(* Logix 5000 project; controller cal1632 1756-L62 rev 16.20; software revision 16.05; part 16 of 61 *)
(* tags used below, declared in another part *)
   FAULT : BOOL;
   HMI : BOOL;
   p01r09_pb_global_reset : BOOL;
   p12_ai_exhaust_amps : REAL;
   p12_ai_exhaust_hz : REAL;
   p12_ai_exhaust_pct : REAL;
   p12_ai_exhaust_rpm : REAL;
   p12_ai_lfl : REAL;
   p12_ai_prs : REAL;
   p12_ai_recirc_amps : REAL;
   p12_ai_recirc_hz : REAL;
   p12_ai_recirc_pct : REAL;
   p12_ai_recirc_rpm : REAL;
   p12_ai_tc01 : REAL;
   p12_ai_tc02 : REAL;
   p12_ao_cv : REAL;
   p12_ao_exhaust_selected_speed : REAL;
   p12_ao_recirc_selected_speed : REAL;
   p12_di_burner_auto : BOOL;
   p12_di_burner_safeties_ok : BOOL;
   p12_di_door_open : BOOL;
   p12_di_exh : acs800_di_normal;
   p12_di_exh_fan_mtr_ts : BOOL;
   p12_di_exh_flow_ok : BOOL;
   p12_di_flame_failure : BOOL;
   p12_di_flame_on : BOOL;
   p12_di_fresh_air_clean : BOOL;
   p12_di_high_limit_temp_ok : BOOL;
   p12_di_recirc : acs800_di_normal;
   p12_di_recirc_fan_mtr_ts : BOOL;
   p12_di_recirc_flow_ok : BOOL;
   p12_di_sp00 : BOOL;
   p12_di_tc01_bo : BOOL;
   p12_di_tc02_bo : BOOL;
   p12_di_zone_air_clean : BOOL;
   p12_dint_to_hmi : DINT[16];
   p12_param_fast_to_soak : REAL;
   p12_param_lfl_hhl : REAL;
   p12_param_lfl_hl : REAL;
   p12_param_pid1_ff : REAL;
   p12_param_pid1_kd : REAL;
   p12_param_pid1_ki : REAL;
   p12_param_pid1_kp : REAL;
   p12_param_pid2_ff : REAL;
   p12_param_pid2_kd : REAL;
   p12_param_pid2_ki : REAL;
   p12_param_pid2_kp : REAL;
   p12_param_shutdown_temp : REAL;
   p12_param_soak_to_fast : REAL;
   p12_param_tc01_dev : REAL;
   p12_param_tc01_hl : REAL;
   p12_param_tc01z : REAL;
   p12_param_tc02z : REAL;
   p12_param_zone_pressure : REAL;
   p12_real_to_hmi : REAL[112];
   p12r05 : routine;
   p12r05_exh_status : DINT;
   p12r05_recirc_status : DINT;
   p12r05_Temp_ctl_status : DINT;
   p12r05_timer_fault : TIMER[4];
   p12r05_timer_warning : TIMER[4];
   p12r06 : routine;
   p12r06_timer_fault : TIMER[4];
   p12r06_timer_warning : TIMER[4];
   p12r07 : routine;
   p12r07_timer_fault : TIMER[4];
   p12r07_timer_warning : TIMER[4];
   p12r20 : routine;
   p12r20_state : DINT;
   p12r20_status : DINT;
   p12r30 : routine;
   p12r30_cv_man_sp : REAL;
   p12r30_permissive_run : BOOL;
   p12r30_pid_temp : PID;
   p12r30_pid_temp_pv : REAL;
   p12r30_pid_temp_sp : REAL;
   p12r30_request_heat : BOOL;
   p12r30_request_manual : BOOL;
   p12r30_vfds_ready : BOOL;
   p12r31 : routine;
   p12r31_request_auto_run : BOOL;
   p12r31_request_auto_stop : BOOL;
   p12r31_vfd_stopped : BOOL;
   p12r32 : routine;
   p12r32_request_auto_run : BOOL;
   p12r32_request_auto_stop : BOOL;
   p12r32_vfd_stopped : BOOL;
(* P12_Zone_2, continued *)

ROUTINE R05_Dint_to_HMI   (* ladder *)
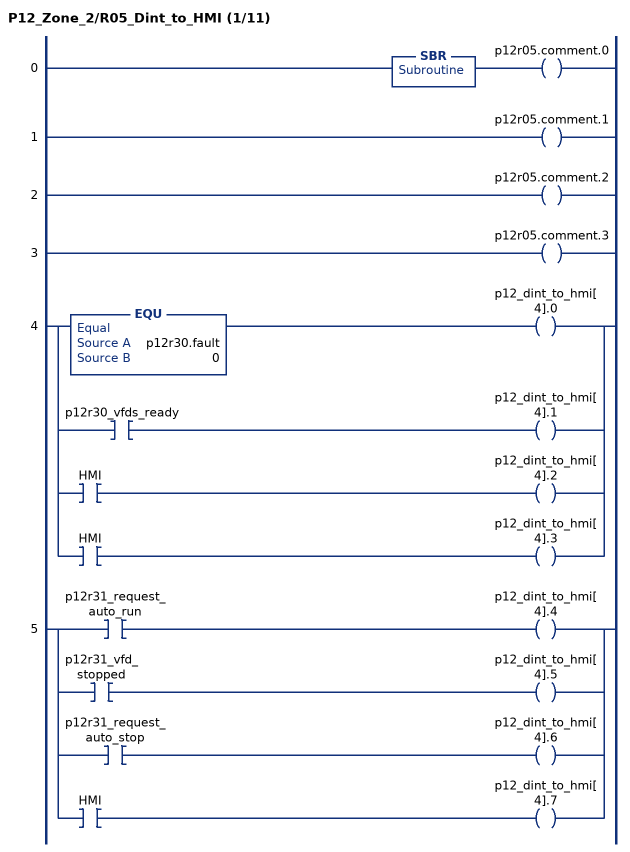
   0: SBR()OTE(p12r05.comment.0);
   1: OTE(p12r05.comment.1);
   2: OTE(p12r05.comment.2);
   3: OTE(p12r05.comment.3);
   4: [EQU(p12r30.fault,0) OTE(p12_dint_to_hmi[4].0) ,XIC(p12r30_vfds_ready) OTE(p12_dint_to_hmi[4].1) ,XIC(HMI) OTE(p12_dint_to_hmi[4].2) ,XIC(HMI) OTE(p12_dint_to_hmi[4].3) ];
   5: [XIC(p12r31_request_auto_run) OTE(p12_dint_to_hmi[4].4) ,XIC(p12r31_vfd_stopped) OTE(p12_dint_to_hmi[4].5) ,XIC(p12r31_request_auto_stop) OTE(p12_dint_to_hmi[4].6) ,XIC(HMI) OTE(p12_dint_to_hmi[4].7) ];
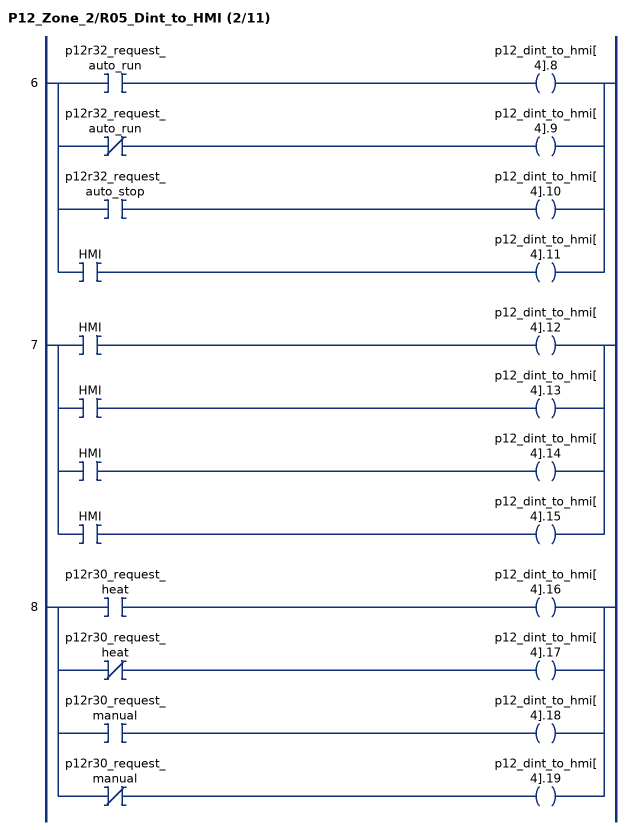
   6: [XIC(p12r32_request_auto_run) OTE(p12_dint_to_hmi[4].8) ,XIO(p12r32_request_auto_run) OTE(p12_dint_to_hmi[4].9) ,XIC(p12r32_request_auto_stop) OTE(p12_dint_to_hmi[4].10) ,XIC(HMI) OTE(p12_dint_to_hmi[4].11) ];
   7: [XIC(HMI) OTE(p12_dint_to_hmi[4].12) ,XIC(HMI) OTE(p12_dint_to_hmi[4].13) ,XIC(HMI) OTE(p12_dint_to_hmi[4].14) ,XIC(HMI) OTE(p12_dint_to_hmi[4].15) ];
   8: [XIC(p12r30_request_heat) OTE(p12_dint_to_hmi[4].16) ,XIO(p12r30_request_heat) OTE(p12_dint_to_hmi[4].17) ,XIC(p12r30_request_manual) OTE(p12_dint_to_hmi[4].18) ,XIO(p12r30_request_manual) OTE(p12_dint_to_hmi[4].19) ];
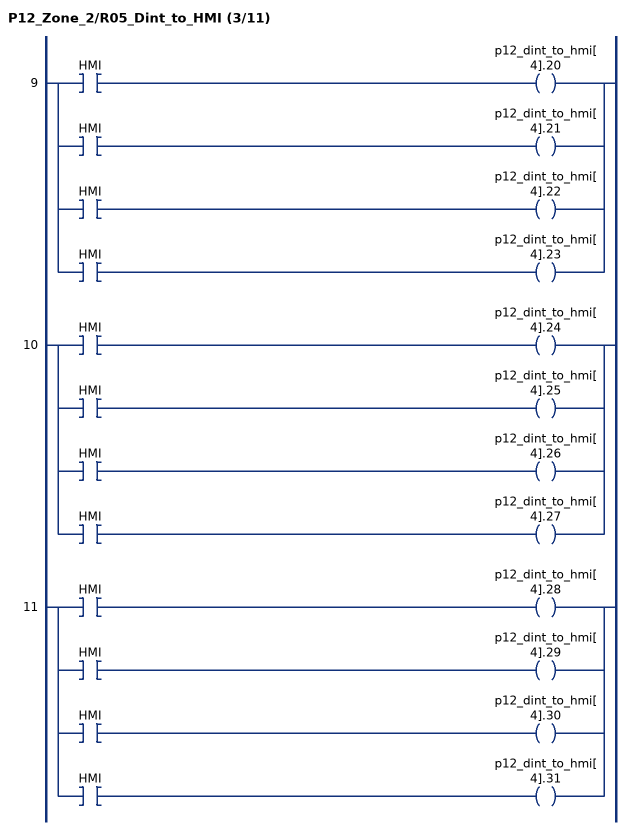
   9: [XIC(HMI) OTE(p12_dint_to_hmi[4].20) ,XIC(HMI) OTE(p12_dint_to_hmi[4].21) ,XIC(HMI) OTE(p12_dint_to_hmi[4].22) ,XIC(HMI) OTE(p12_dint_to_hmi[4].23) ];
   10: [XIC(HMI) OTE(p12_dint_to_hmi[4].24) ,XIC(HMI) OTE(p12_dint_to_hmi[4].25) ,XIC(HMI) OTE(p12_dint_to_hmi[4].26) ,XIC(HMI) OTE(p12_dint_to_hmi[4].27) ];
   11: [XIC(HMI) OTE(p12_dint_to_hmi[4].28) ,XIC(HMI) OTE(p12_dint_to_hmi[4].29) ,XIC(HMI) OTE(p12_dint_to_hmi[4].30) ,XIC(HMI) OTE(p12_dint_to_hmi[4].31) ];
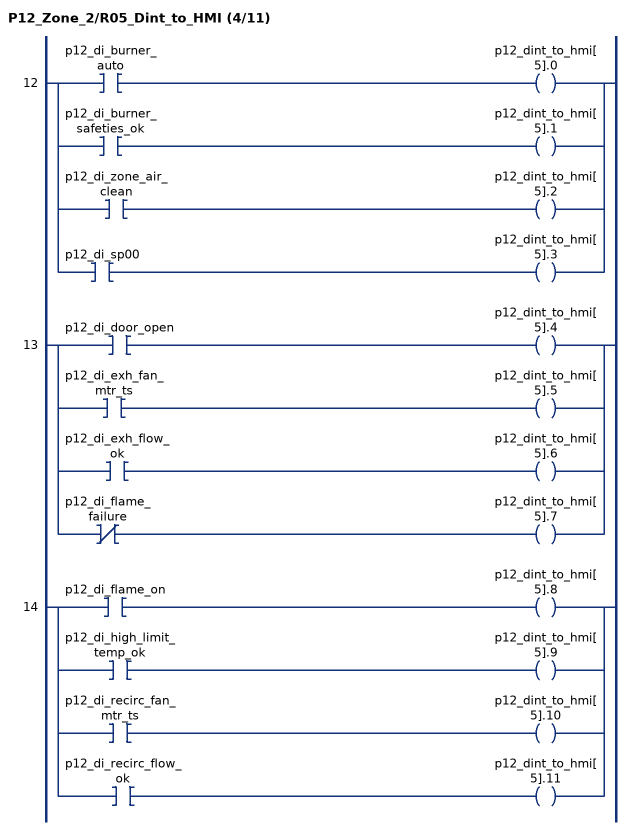
   12: [XIC(p12_di_burner_auto) OTE(p12_dint_to_hmi[5].0) ,XIC(p12_di_burner_safeties_ok) OTE(p12_dint_to_hmi[5].1) ,XIC(p12_di_zone_air_clean) OTE(p12_dint_to_hmi[5].2) ,XIC(p12_di_sp00) OTE(p12_dint_to_hmi[5].3) ];
   13: [XIC(p12_di_door_open) OTE(p12_dint_to_hmi[5].4) ,XIC(p12_di_exh_fan_mtr_ts) OTE(p12_dint_to_hmi[5].5) ,XIC(p12_di_exh_flow_ok) OTE(p12_dint_to_hmi[5].6) ,XIO(p12_di_flame_failure) OTE(p12_dint_to_hmi[5].7) ];
   14: [XIC(p12_di_flame_on) OTE(p12_dint_to_hmi[5].8) ,XIC(p12_di_high_limit_temp_ok) OTE(p12_dint_to_hmi[5].9) ,XIC(p12_di_recirc_fan_mtr_ts) OTE(p12_dint_to_hmi[5].10) ,XIC(p12_di_recirc_flow_ok) OTE(p12_dint_to_hmi[5].11) ];
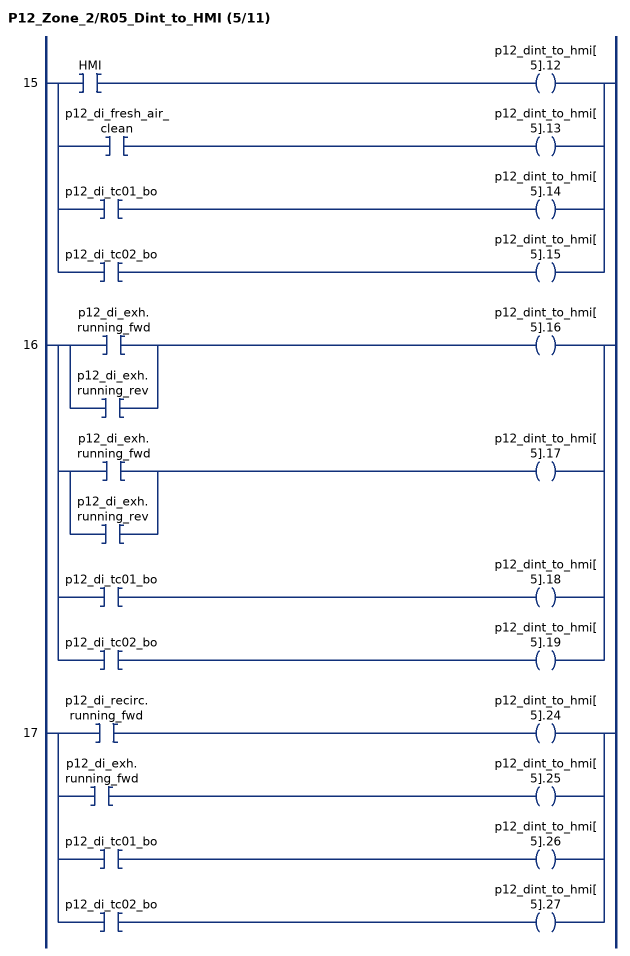
   15: [XIC(HMI) OTE(p12_dint_to_hmi[5].12) ,XIC(p12_di_fresh_air_clean) OTE(p12_dint_to_hmi[5].13) ,XIC(p12_di_tc01_bo) OTE(p12_dint_to_hmi[5].14) ,XIC(p12_di_tc02_bo) OTE(p12_dint_to_hmi[5].15) ];
   16: [[XIC(p12_di_exh.running_fwd) ,XIC(p12_di_exh.running_rev) ] OTE(p12_dint_to_hmi[5].16) ,[XIC(p12_di_exh.running_fwd) ,XIC(p12_di_exh.running_rev) ] OTE(p12_dint_to_hmi[5].17) ,XIC(p12_di_tc01_bo) OTE(p12_dint_to_hmi[5].18) ,XIC(p12_di_tc02_bo) OTE(p12_dint_to_hmi[5].19) ];
   17: [XIC(p12_di_recirc.running_fwd) OTE(p12_dint_to_hmi[5].24) ,XIC(p12_di_exh.running_fwd) OTE(p12_dint_to_hmi[5].25) ,XIC(p12_di_tc01_bo) OTE(p12_dint_to_hmi[5].26) ,XIC(p12_di_tc02_bo) OTE(p12_dint_to_hmi[5].27) ];
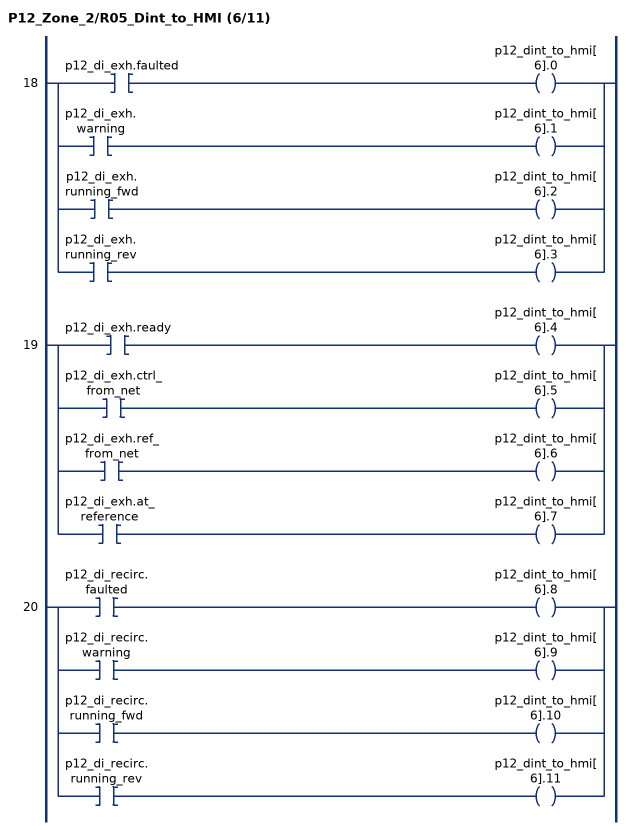
   18: [XIC(p12_di_exh.faulted) OTE(p12_dint_to_hmi[6].0) ,XIC(p12_di_exh.warning) OTE(p12_dint_to_hmi[6].1) ,XIC(p12_di_exh.running_fwd) OTE(p12_dint_to_hmi[6].2) ,XIC(p12_di_exh.running_rev) OTE(p12_dint_to_hmi[6].3) ];
   19: [XIC(p12_di_exh.ready) OTE(p12_dint_to_hmi[6].4) ,XIC(p12_di_exh.ctrl_from_net) OTE(p12_dint_to_hmi[6].5) ,XIC(p12_di_exh.ref_from_net) OTE(p12_dint_to_hmi[6].6) ,XIC(p12_di_exh.at_reference) OTE(p12_dint_to_hmi[6].7) ];
   20: [XIC(p12_di_recirc.faulted) OTE(p12_dint_to_hmi[6].8) ,XIC(p12_di_recirc.warning) OTE(p12_dint_to_hmi[6].9) ,XIC(p12_di_recirc.running_fwd) OTE(p12_dint_to_hmi[6].10) ,XIC(p12_di_recirc.running_rev) OTE(p12_dint_to_hmi[6].11) ];
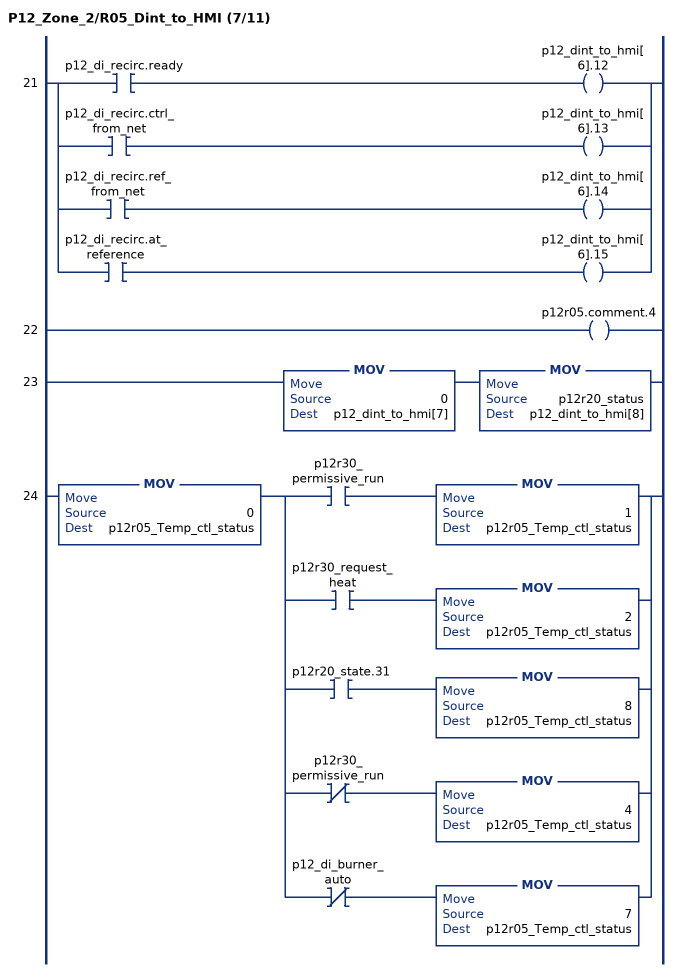
   21: [XIC(p12_di_recirc.ready) OTE(p12_dint_to_hmi[6].12) ,XIC(p12_di_recirc.ctrl_from_net) OTE(p12_dint_to_hmi[6].13) ,XIC(p12_di_recirc.ref_from_net) OTE(p12_dint_to_hmi[6].14) ,XIC(p12_di_recirc.at_reference) OTE(p12_dint_to_hmi[6].15) ];
   22: OTE(p12r05.comment.4);
   23: MOV(0,p12_dint_to_hmi[7])MOV(p12r20_status,p12_dint_to_hmi[8]);
   24: MOV(0,p12r05_Temp_ctl_status)[XIC(p12r30_permissive_run) MOV(1,p12r05_Temp_ctl_status) ,XIC(p12r30_request_heat) MOV(2,p12r05_Temp_ctl_status) ,XIC(p12r20_state.31) MOV(8,p12r05_Temp_ctl_status) ,XIO(p12r30_permissive_run) MOV(4,p12r05_Temp_ctl_status) ,XIO(p12_di_burner_auto) MOV(7,p12r05_Temp_ctl_status) ];
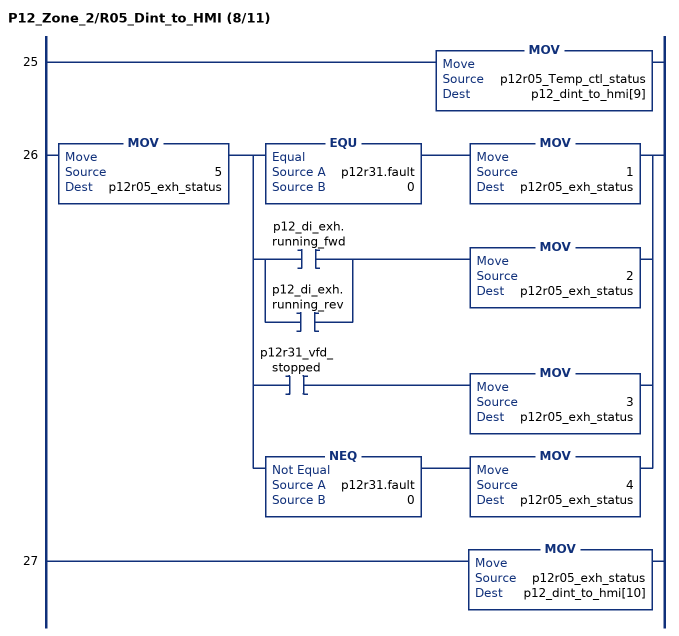
   25: MOV(p12r05_Temp_ctl_status,p12_dint_to_hmi[9]);
   26: MOV(5,p12r05_exh_status)[EQU(p12r31.fault,0) MOV(1,p12r05_exh_status) ,[XIC(p12_di_exh.running_fwd) ,XIC(p12_di_exh.running_rev) ] MOV(2,p12r05_exh_status) ,XIC(p12r31_vfd_stopped) MOV(3,p12r05_exh_status) ,NEQ(p12r31.fault,0) MOV(4,p12r05_exh_status) ];
   27: MOV(p12r05_exh_status,p12_dint_to_hmi[10]);
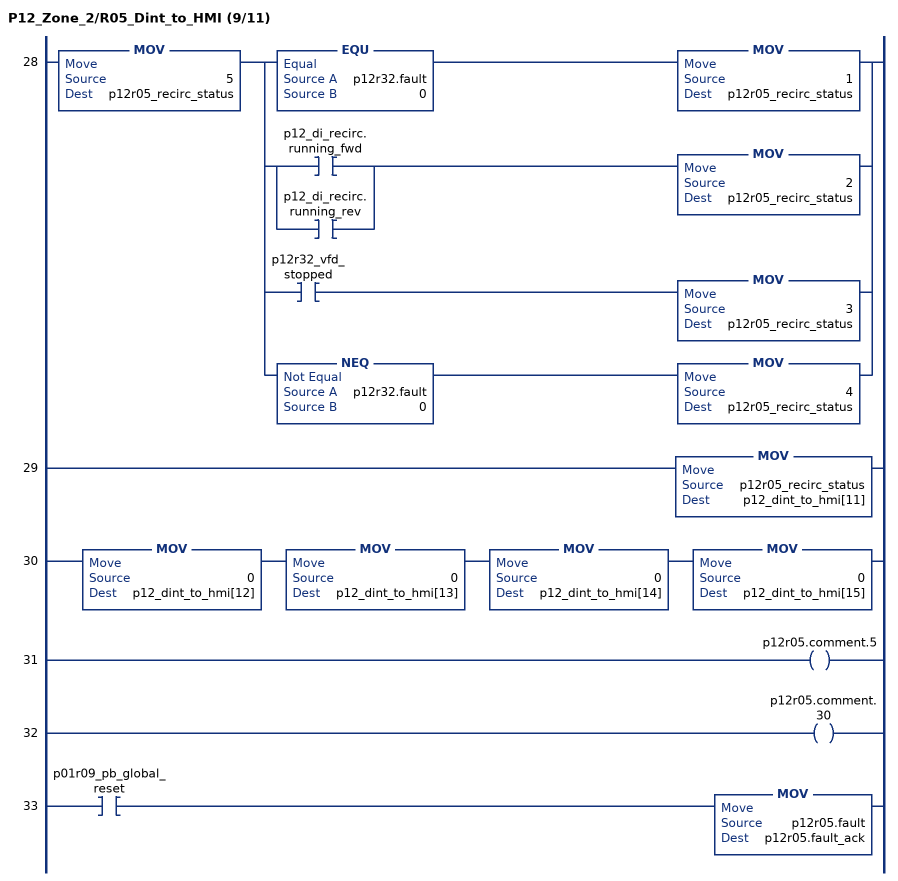
   28: MOV(5,p12r05_recirc_status)[EQU(p12r32.fault,0) MOV(1,p12r05_recirc_status) ,[XIC(p12_di_recirc.running_fwd) ,XIC(p12_di_recirc.running_rev) ] MOV(2,p12r05_recirc_status) ,XIC(p12r32_vfd_stopped) MOV(3,p12r05_recirc_status) ,NEQ(p12r32.fault,0) MOV(4,p12r05_recirc_status) ];
   29: MOV(p12r05_recirc_status,p12_dint_to_hmi[11]);
   30: MOV(0,p12_dint_to_hmi[12])MOV(0,p12_dint_to_hmi[13])MOV(0,p12_dint_to_hmi[14])MOV(0,p12_dint_to_hmi[15]);
   31: OTE(p12r05.comment.5);
   32: OTE(p12r05.comment.30);
   33: XIC(p01r09_pb_global_reset)MOV(p12r05.fault,p12r05.fault_ack);
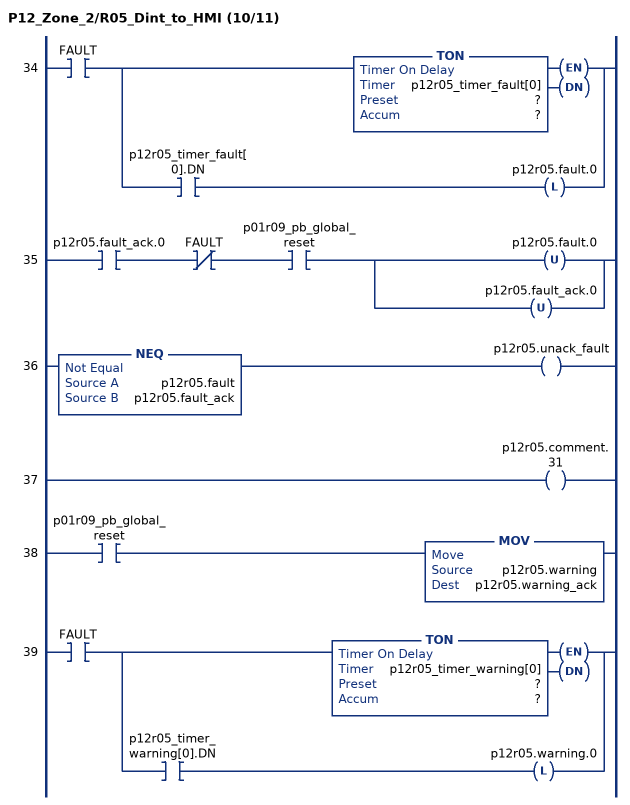
   34: XIC(FAULT)[TON(p12r05_timer_fault[0],?,?) ,XIC(p12r05_timer_fault[0].DN) OTL(p12r05.fault.0) ];
   35: XIC(p12r05.fault_ack.0)XIO(FAULT)XIC(p01r09_pb_global_reset)[OTU(p12r05.fault.0) ,OTU(p12r05.fault_ack.0) ];
   36: NEQ(p12r05.fault,p12r05.fault_ack)OTE(p12r05.unack_fault);
   37: OTE(p12r05.comment.31);
   38: XIC(p01r09_pb_global_reset)MOV(p12r05.warning,p12r05.warning_ack);
   39: XIC(FAULT)[TON(p12r05_timer_warning[0],?,?) ,XIC(p12r05_timer_warning[0].DN) OTL(p12r05.warning.0) ];
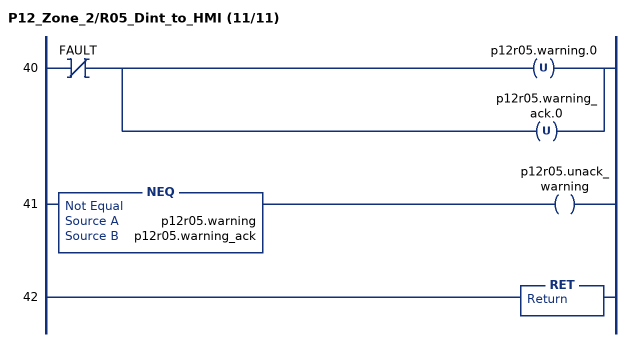
   40: XIO(FAULT)[OTU(p12r05.warning.0) ,OTU(p12r05.warning_ack.0) ];
   41: NEQ(p12r05.warning,p12r05.warning_ack)OTE(p12r05.unack_warning);
   42: RET();
END_ROUTINE

ROUTINE R06_Real_to_HMI   (* ladder *)
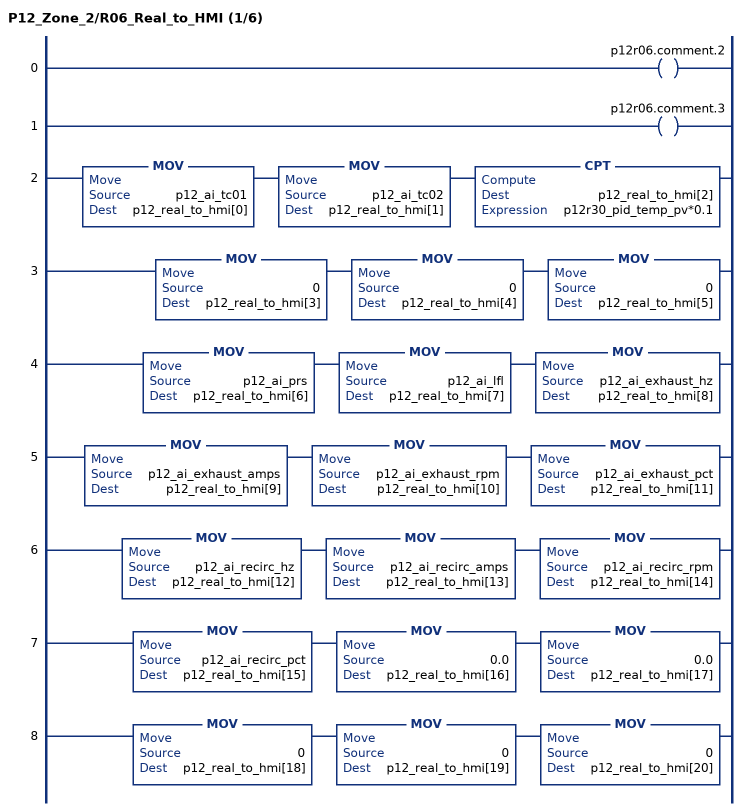
   0: OTE(p12r06.comment.2);
   1: OTE(p12r06.comment.3);
   2: MOV(p12_ai_tc01,p12_real_to_hmi[0])MOV(p12_ai_tc02,p12_real_to_hmi[1])CPT(p12_real_to_hmi[2],p12r30_pid_temp_pv*0.1);
   3: MOV(0,p12_real_to_hmi[3])MOV(0,p12_real_to_hmi[4])MOV(0,p12_real_to_hmi[5]);
   4: MOV(p12_ai_prs,p12_real_to_hmi[6])MOV(p12_ai_lfl,p12_real_to_hmi[7])MOV(p12_ai_exhaust_hz,p12_real_to_hmi[8]);
   5: MOV(p12_ai_exhaust_amps,p12_real_to_hmi[9])MOV(p12_ai_exhaust_rpm,p12_real_to_hmi[10])MOV(p12_ai_exhaust_pct,p12_real_to_hmi[11]);
   6: MOV(p12_ai_recirc_hz,p12_real_to_hmi[12])MOV(p12_ai_recirc_amps,p12_real_to_hmi[13])MOV(p12_ai_recirc_rpm,p12_real_to_hmi[14]);
   7: MOV(p12_ai_recirc_pct,p12_real_to_hmi[15])MOV(0.0,p12_real_to_hmi[16])MOV(0.0,p12_real_to_hmi[17]);
   8: MOV(0,p12_real_to_hmi[18])MOV(0,p12_real_to_hmi[19])MOV(0,p12_real_to_hmi[20]);
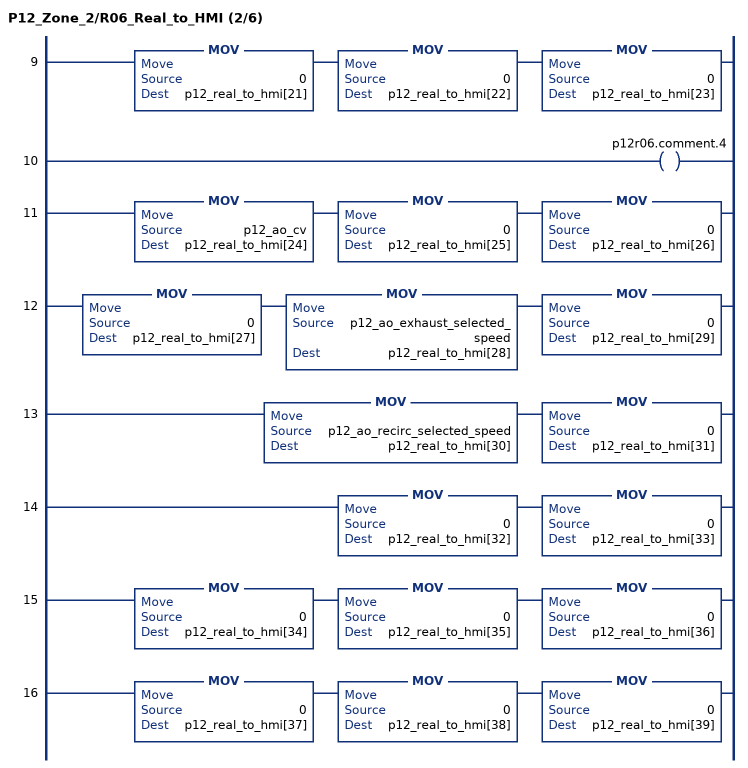
   9: MOV(0,p12_real_to_hmi[21])MOV(0,p12_real_to_hmi[22])MOV(0,p12_real_to_hmi[23]);
   10: OTE(p12r06.comment.4);
   11: MOV(p12_ao_cv,p12_real_to_hmi[24])MOV(0,p12_real_to_hmi[25])MOV(0,p12_real_to_hmi[26]);
   12: MOV(0,p12_real_to_hmi[27])MOV(p12_ao_exhaust_selected_speed,p12_real_to_hmi[28])MOV(0,p12_real_to_hmi[29]);
   13: MOV(p12_ao_recirc_selected_speed,p12_real_to_hmi[30])MOV(0,p12_real_to_hmi[31]);
   14: MOV(0,p12_real_to_hmi[32])MOV(0,p12_real_to_hmi[33]);
   15: MOV(0,p12_real_to_hmi[34])MOV(0,p12_real_to_hmi[35])MOV(0,p12_real_to_hmi[36]);
   16: MOV(0,p12_real_to_hmi[37])MOV(0,p12_real_to_hmi[38])MOV(0,p12_real_to_hmi[39]);
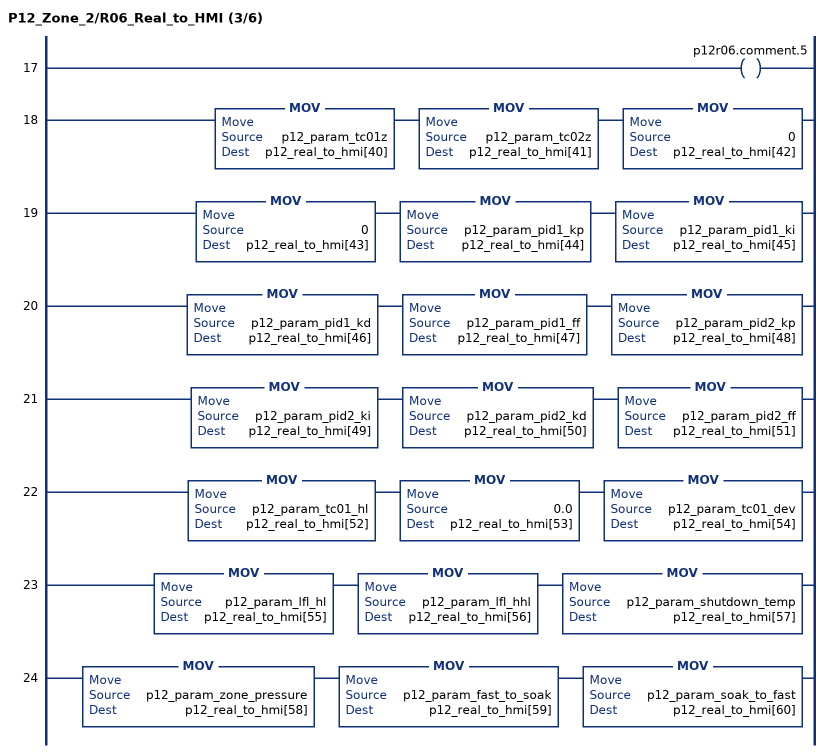
   17: OTE(p12r06.comment.5);
   18: MOV(p12_param_tc01z,p12_real_to_hmi[40])MOV(p12_param_tc02z,p12_real_to_hmi[41])MOV(0,p12_real_to_hmi[42]);
   19: MOV(0,p12_real_to_hmi[43])MOV(p12_param_pid1_kp,p12_real_to_hmi[44])MOV(p12_param_pid1_ki,p12_real_to_hmi[45]);
   20: MOV(p12_param_pid1_kd,p12_real_to_hmi[46])MOV(p12_param_pid1_ff,p12_real_to_hmi[47])MOV(p12_param_pid2_kp,p12_real_to_hmi[48]);
   21: MOV(p12_param_pid2_ki,p12_real_to_hmi[49])MOV(p12_param_pid2_kd,p12_real_to_hmi[50])MOV(p12_param_pid2_ff,p12_real_to_hmi[51]);
   22: MOV(p12_param_tc01_hl,p12_real_to_hmi[52])MOV(0.0,p12_real_to_hmi[53])MOV(p12_param_tc01_dev,p12_real_to_hmi[54]);
   23: MOV(p12_param_lfl_hl,p12_real_to_hmi[55])MOV(p12_param_lfl_hhl,p12_real_to_hmi[56])MOV(p12_param_shutdown_temp,p12_real_to_hmi[57]);
   24: MOV(p12_param_zone_pressure,p12_real_to_hmi[58])MOV(p12_param_fast_to_soak,p12_real_to_hmi[59])MOV(p12_param_soak_to_fast,p12_real_to_hmi[60]);
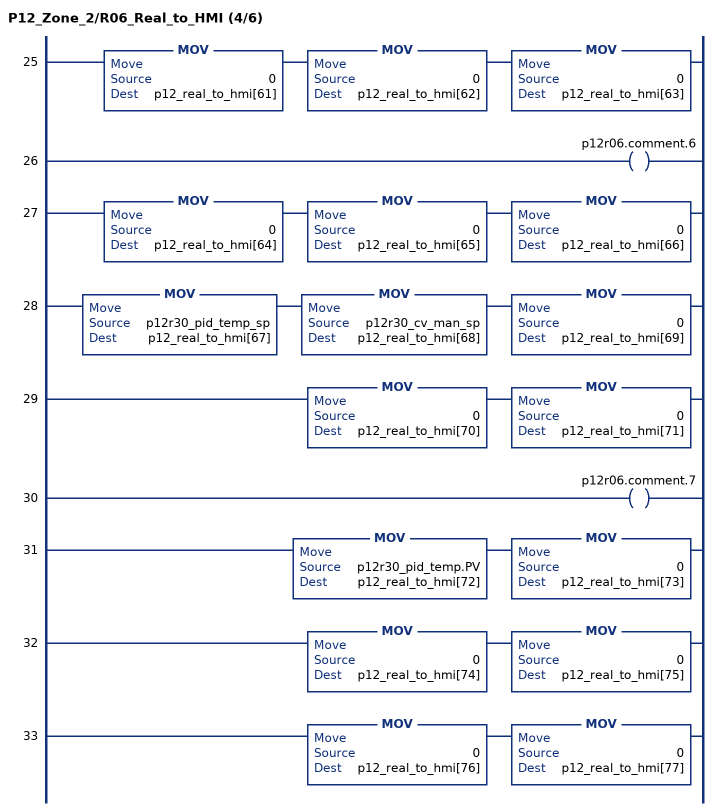
   25: MOV(0,p12_real_to_hmi[61])MOV(0,p12_real_to_hmi[62])MOV(0,p12_real_to_hmi[63]);
   26: OTE(p12r06.comment.6);
   27: MOV(0,p12_real_to_hmi[64])MOV(0,p12_real_to_hmi[65])MOV(0,p12_real_to_hmi[66]);
   28: MOV(p12r30_pid_temp_sp,p12_real_to_hmi[67])MOV(p12r30_cv_man_sp,p12_real_to_hmi[68])MOV(0,p12_real_to_hmi[69]);
   29: MOV(0,p12_real_to_hmi[70])MOV(0,p12_real_to_hmi[71]);
   30: OTE(p12r06.comment.7);
   31: MOV(p12r30_pid_temp.PV,p12_real_to_hmi[72])MOV(0,p12_real_to_hmi[73]);
   32: MOV(0,p12_real_to_hmi[74])MOV(0,p12_real_to_hmi[75]);
   33: MOV(0,p12_real_to_hmi[76])MOV(0,p12_real_to_hmi[77]);
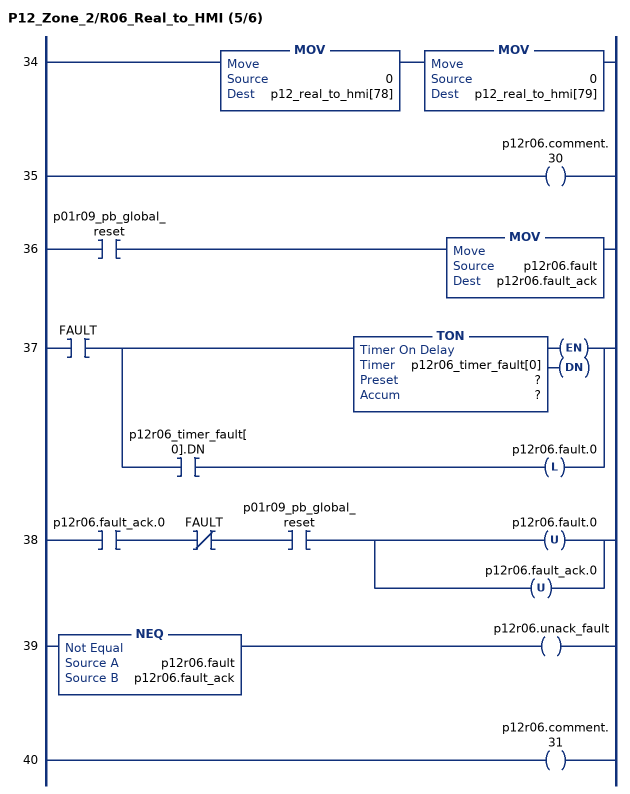
   34: MOV(0,p12_real_to_hmi[78])MOV(0,p12_real_to_hmi[79]);
   35: OTE(p12r06.comment.30);
   36: XIC(p01r09_pb_global_reset)MOV(p12r06.fault,p12r06.fault_ack);
   37: XIC(FAULT)[TON(p12r06_timer_fault[0],?,?) ,XIC(p12r06_timer_fault[0].DN) OTL(p12r06.fault.0) ];
   38: XIC(p12r06.fault_ack.0)XIO(FAULT)XIC(p01r09_pb_global_reset)[OTU(p12r06.fault.0) ,OTU(p12r06.fault_ack.0) ];
   39: NEQ(p12r06.fault,p12r06.fault_ack)OTE(p12r06.unack_fault);
   40: OTE(p12r06.comment.31);
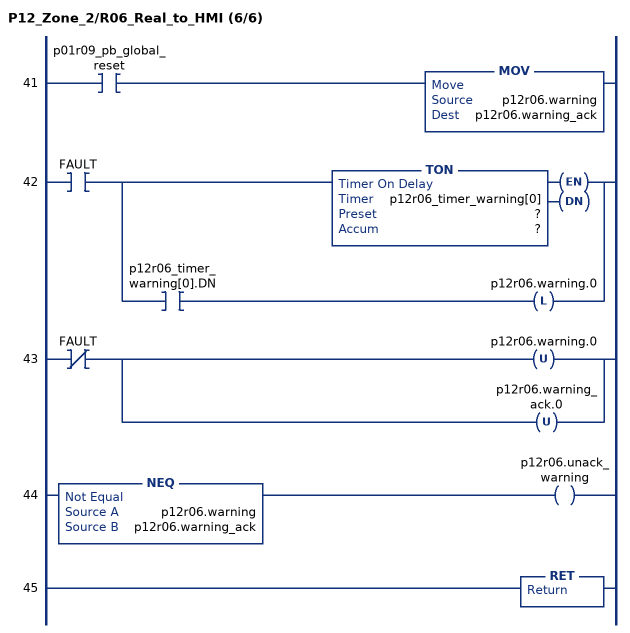
   41: XIC(p01r09_pb_global_reset)MOV(p12r06.warning,p12r06.warning_ack);
   42: XIC(FAULT)[TON(p12r06_timer_warning[0],?,?) ,XIC(p12r06_timer_warning[0].DN) OTL(p12r06.warning.0) ];
   43: XIO(FAULT)[OTU(p12r06.warning.0) ,OTU(p12r06.warning_ack.0) ];
   44: NEQ(p12r06.warning,p12r06.warning_ack)OTE(p12r06.unack_warning);
   45: RET();
END_ROUTINE

ROUTINE R07_Alarms   (* ladder *)
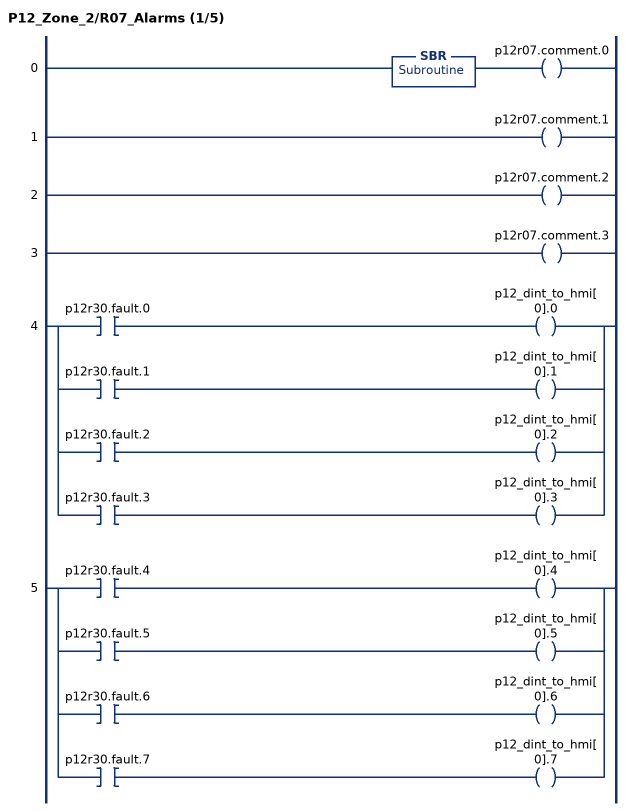
   0: SBR()OTE(p12r07.comment.0);
   1: OTE(p12r07.comment.1);
   2: OTE(p12r07.comment.2);
   3: OTE(p12r07.comment.3);
   4: [XIC(p12r30.fault.0) OTE(p12_dint_to_hmi[0].0) ,XIC(p12r30.fault.1) OTE(p12_dint_to_hmi[0].1) ,XIC(p12r30.fault.2) OTE(p12_dint_to_hmi[0].2) ,XIC(p12r30.fault.3) OTE(p12_dint_to_hmi[0].3) ];
   5: [XIC(p12r30.fault.4) OTE(p12_dint_to_hmi[0].4) ,XIC(p12r30.fault.5) OTE(p12_dint_to_hmi[0].5) ,XIC(p12r30.fault.6) OTE(p12_dint_to_hmi[0].6) ,XIC(p12r30.fault.7) OTE(p12_dint_to_hmi[0].7) ];
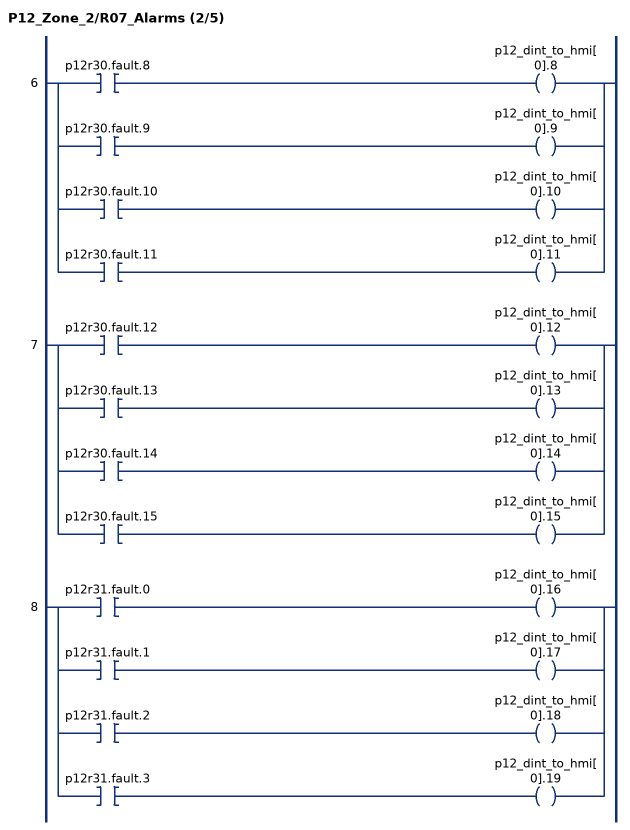
   6: [XIC(p12r30.fault.8) OTE(p12_dint_to_hmi[0].8) ,XIC(p12r30.fault.9) OTE(p12_dint_to_hmi[0].9) ,XIC(p12r30.fault.10) OTE(p12_dint_to_hmi[0].10) ,XIC(p12r30.fault.11) OTE(p12_dint_to_hmi[0].11) ];
   7: [XIC(p12r30.fault.12) OTE(p12_dint_to_hmi[0].12) ,XIC(p12r30.fault.13) OTE(p12_dint_to_hmi[0].13) ,XIC(p12r30.fault.14) OTE(p12_dint_to_hmi[0].14) ,XIC(p12r30.fault.15) OTE(p12_dint_to_hmi[0].15) ];
   8: [XIC(p12r31.fault.0) OTE(p12_dint_to_hmi[0].16) ,XIC(p12r31.fault.1) OTE(p12_dint_to_hmi[0].17) ,XIC(p12r31.fault.2) OTE(p12_dint_to_hmi[0].18) ,XIC(p12r31.fault.3) OTE(p12_dint_to_hmi[0].19) ];
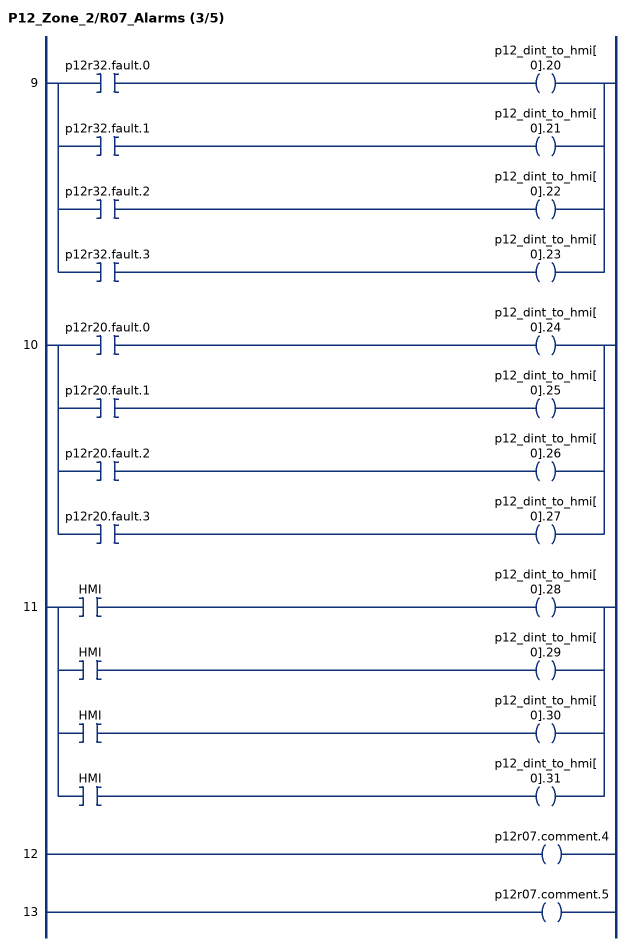
   9: [XIC(p12r32.fault.0) OTE(p12_dint_to_hmi[0].20) ,XIC(p12r32.fault.1) OTE(p12_dint_to_hmi[0].21) ,XIC(p12r32.fault.2) OTE(p12_dint_to_hmi[0].22) ,XIC(p12r32.fault.3) OTE(p12_dint_to_hmi[0].23) ];
   10: [XIC(p12r20.fault.0) OTE(p12_dint_to_hmi[0].24) ,XIC(p12r20.fault.1) OTE(p12_dint_to_hmi[0].25) ,XIC(p12r20.fault.2) OTE(p12_dint_to_hmi[0].26) ,XIC(p12r20.fault.3) OTE(p12_dint_to_hmi[0].27) ];
   11: [XIC(HMI) OTE(p12_dint_to_hmi[0].28) ,XIC(HMI) OTE(p12_dint_to_hmi[0].29) ,XIC(HMI) OTE(p12_dint_to_hmi[0].30) ,XIC(HMI) OTE(p12_dint_to_hmi[0].31) ];
   12: OTE(p12r07.comment.4);
   13: OTE(p12r07.comment.5);
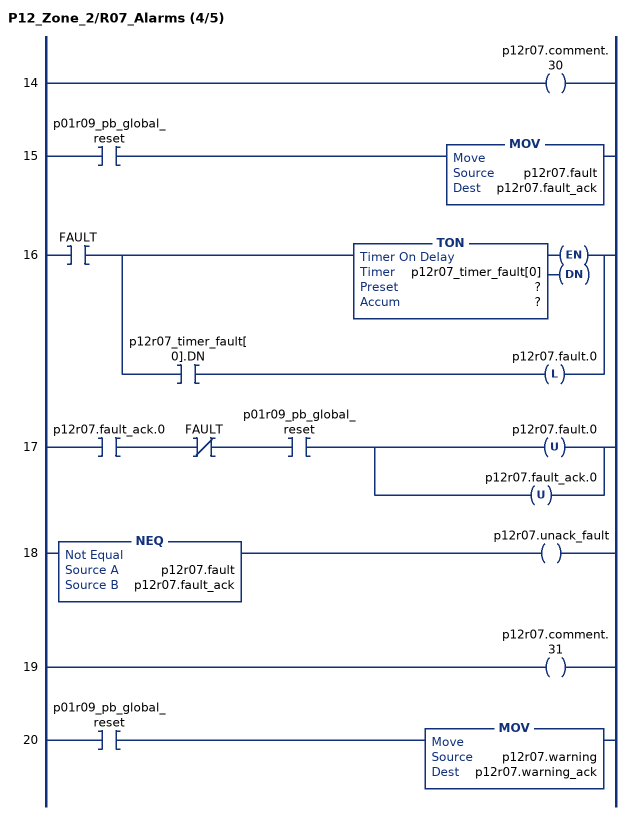
   14: OTE(p12r07.comment.30);
   15: XIC(p01r09_pb_global_reset)MOV(p12r07.fault,p12r07.fault_ack);
   16: XIC(FAULT)[TON(p12r07_timer_fault[0],?,?) ,XIC(p12r07_timer_fault[0].DN) OTL(p12r07.fault.0) ];
   17: XIC(p12r07.fault_ack.0)XIO(FAULT)XIC(p01r09_pb_global_reset)[OTU(p12r07.fault.0) ,OTU(p12r07.fault_ack.0) ];
   18: NEQ(p12r07.fault,p12r07.fault_ack)OTE(p12r07.unack_fault);
   19: OTE(p12r07.comment.31);
   20: XIC(p01r09_pb_global_reset)MOV(p12r07.warning,p12r07.warning_ack);
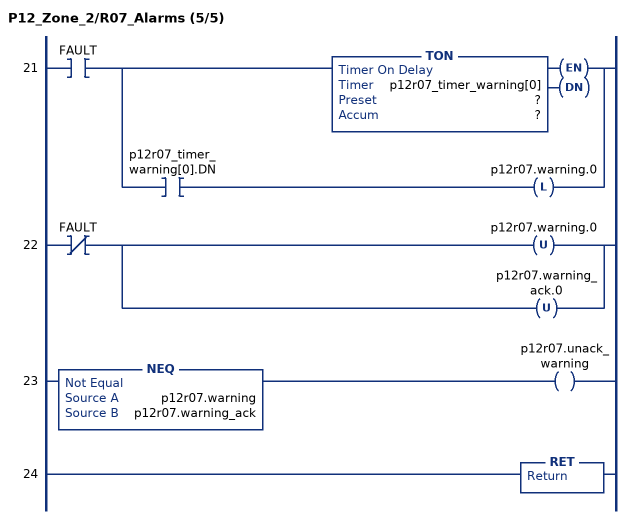
   21: XIC(FAULT)[TON(p12r07_timer_warning[0],?,?) ,XIC(p12r07_timer_warning[0].DN) OTL(p12r07.warning.0) ];
   22: XIO(FAULT)[OTU(p12r07.warning.0) ,OTU(p12r07.warning_ack.0) ];
   23: NEQ(p12r07.warning,p12r07.warning_ack)OTE(p12r07.unack_warning);
   24: RET();
END_ROUTINE
